(* IEC 61131-3 sources: verifaps-lib/iec-symbex/src/test/resources/edu/kit/iti/formal/automation, 3 files *)

(* ---- fbembedding_1.st ---- *)
PROGRAM main
VAR_INPUT i : INT; END_VAR
VAR_OUTPUT o : INT; END_VAR

VAR
   a : FB1;
END_VAR
a(j:=i);
o:=a.p;
END_PROGRAM

FUNCTION_BLOCK FB1

VAR_INPUT j : INT; END_VAR
VAR_OUTPUT p : INT; END_VAR
VAR sum : INT; END_VAR

sum := p + sum;
p := sum / p;

END_FUNCTION_BLOCK

(* ---- program_with_actions.st ---- *)
PROGRAM abc
    VAR_INPUT
        i : INT;
    END_VAR
    VAR_OUTPUT
        o : INT;
    END_VAR
    VAR
        s: INT;
    END_VAR

    ACTION up
        s := s + i;
    END_ACTION

    ACTION down
        s := s - i;
    END_ACTION

    IF i < 0 THEN
        down();
    ELSE
        up();
    END_IF
    o:=s;
END_PROGRAM

(* ---- struct_embedding.st ---- *)
TYPE
  A: STRUCT
    x : INT;
    y : INT;
  END_STRUCT;
END_TYPE

FUNCTION g : INT
  VAR_INPUT
    a : A;
  END_VAR

  g := a.x + a.y;
END_FUNCTION

FUNCTION A_f : INT
  VAR_INPUT
    _SELF : A;
    z : INT;
  END_VAR

  IF (_SELF.x > z) THEN
    A_f := _SELF.y;
  ELSE
    A_f := z;
  END_IF
END_FUNCTION

PROGRAM MY_PROGRAM
  VAR_INPUT
    z : INT;
  END_VAR
  VAR
    a : A := (x := 42, y := 333);
  END_VAR
  VAR_OUTPUT
    new_z : INT;
  END_VAR

  new_z := A_f(_SELF := a, z := z) + g(a);
END_PROGRAM
